// TIA Portal V17 export
// export: Created 2025-03-10T13:12:17.8643549Z, ExportSetting WithDefaults, DisplayName Totally Integrated Automation Portal, DisplayVersion V17 Update 8, DisplayName TIA Portal Openness, DisplayVersion V17 Update 8, DisplayName TIA Portal Version Control Interface, DisplayVersion V17, DisplayName SINAMICS Startdrive Advanced, DisplayVersion V17 SP2, DisplayName SINAMICS Startdrive G110M, G120, G120C, G120D, G120P, G115D, DisplayVersion V17 SP2, DisplayName SINAMICS Startdrive G130, G150, S120, S150, SINAMICS MV, S210, DisplayVersion V17 SP2, DisplayName STEP 7 Professional, DisplayVersion V17 Update 8, DisplayName SINUMERIK ONE STEP 7 Toolbox, DisplayVersion V17 Update 12, DisplayName SINUMERIK 840D sl STEP 7 Toolbox, DisplayVersion V17 Update 12, DisplayName STEP 7 Safety, DisplayVersion V17 Update 6, DisplayName WinCC Advanced, DisplayVersion V17 Update 8
TYPE "FANUC_INPUTS"
// stored: IsFailsafeCompliant false
   STRUCT
      SYSTEM_SIGNAL : Struct
         SYS_IMSTP : Bool;   // MACHINE HEARTBEAT (MACHINE TO GANTRY) / IMMEDIATE STOP
         SYS_HOLD : Bool;   // HOLD ROBOT
         SYS_SFSPD : Bool;   // MACHINE EMERGENCY STOP OK (MACHINE TO GANTRY) / SAFE SPEED
         SYS_CYCLE_STOP : Bool;   // MACHINE SAFETY GATES OK (LOCKED)(MACHINE TO GANTRY) / CYCLE STOP
         SYS_FAULT_RESET : Bool;   // MACHINE IN MANUAL MODE (MACHINE TO GANTRY) / FAULT RESET
         SYS_HOME : Bool;   // MACHINE IN AUTO MODE(MACHINE TO GANTRY) / HOME
         SYS_START : Bool;   // MACHINE AUTO CYCLE RUNNING (MACHINE TO GANTRY) / START PROGRAM / CONTINUE PROGRAM
         SYS_MOTION_ENBL : Bool;   // MACHINE IS IN WARMUP CYCLE (MACHINE TO GANTRY) / MOTION ENABLE
         SPARE_65_0 : Byte;   // MACHINE IN RUN OUT MODE (MACHINE TO GANTRY)
         SPARE_66_0 : Byte;   // MACHINE PART DEMAND SOON (MACHINE TO GANTRY)
         SPARE_67_0 : Byte;
      END_STRUCT;
      GENERAL_SIGNAL : Struct
         STYLE_INIT : Bool;   // GANTRY HEARTBEAT (GANTRY TO MACHINE) / INITIATE STYLE PROGRAM
         READ_DEC_CODE : Bool;   // READ DECISION CODE
         OK_CONTINUE : Bool;   // GANTRY EMERGENCY STOP OK (GANTRY TO MACHINE) / OK TO CONTINUE
         ENTER_REQUEST : Bool;   // ENTER CELL REQUEST
         DRY_CYCLE : Bool;   // GANTRY IN MANUAL MODE (GANTRY TO MACHINE) / DRY CYCLE
         RECOVER_REQ : Bool;   // GANTRY IN AUTO MODE (GANTRY TO MACHINE) / RECOVERY REQUEST
         SPARE_68_6 : Bool;   // GANTRY IN AUTO CYCLE RUNNING (GANTRY TO MACHINE)
         SPARE_68_7 : Bool;   // GANTRY OVERHEAD DOOR CLOSED & LOCKED (GANTRY TO MACHINE)
         IMMEDIATE_STOP_AUX : Bool;
         STOP_END_OF_CYCLE : Bool;
         RUNOUT_REQUEST : Bool;
         SPARE_69_3 : Bool;
         SPARE_69_4 : Bool;
         SPARE_69_5 : Bool;
         SPARE_69_6 : Bool;
         SPARE_69_7 : Bool;
         SPARE_70_0 : Byte;   // GANTRY CLEAR OF MACHINE (GANTRY TO MACHINE)
         SPARE_71_0 : Byte;   // GANTRY CLEAR OF FIXTURE (GANTRY TO MACHINE)
         SPARE_72_0 : Byte;
         SPARE_73_0 : Byte;
      END_STRUCT;
      PROGRAM : Struct
         STYLE_PROGRAM : Byte;   // GANTRY HEARTBEAT (GANTRY TO MACHINE) / GROUP INPUT INDICATING STYLE NUMBER PROGRAM
         DEC_CODE : Byte;   // SPECIFIC OPERATING WITHIN A STYLE
         PART_TYPE : Byte;   // GANTRY EMERGENCY STOP OK (GANTRY TO MACHINE) / PART TYPE SELECTED
         SPARE_77_0 : Byte;   // GANTRY EMERGENCY STOP OK (GANTRY TO MACHINE)
      END_STRUCT;
      GRIPPERS : Struct
         T1_GRIPPER_A_OPEN_REQ : Bool;   // ROBOT TOOL 1 GRIPPER A OPEN REQUEST
         T1_GRIPPER_A_CLOSE_REQ : Bool;   // ROBOT TOOL 1 GRIPPER A CLOSE REQUEST
         SPARE_78_2 : Bool;
         SPARE_78_3 : Bool;
         T1_GRIPPER_A_OPEN : Bool;   // ROBOT TOOL 1 GRIPPER A OPEN
         T1_GRIPPER_A_CLOSED : Bool;   // ROBOT TOOL 1 GRIPPER A CLOSED
         SPARE_78_6 : Bool;
         SPARE_78_7 : Bool;
         T1_GRIPPER_B_OPEN_REQ : Bool;   // ROBOT TOOL 1 GRIPPER B OPEN REQUEST
         T1_GRIPPER_B_CLOSE_REQ : Bool;   // ROBOT TOOL 1 GRIPPER B CLOSE REQUEST
         SPARE_79_2 : Bool;
         SPARE_79_3 : Bool;
         T1_GRIPPER_B_OPEN : Bool;   // ROBOT TOOL 1 GRIPPER B OPEN
         T1_GRIPPER_B_CLOSED : Bool;   // ROBOT TOOL 1 GRIPPER B CLOSED
         SPARE_79_6 : Bool;
         SPARE_79_7 : Bool;
         T1_GRIPPER_C_OPEN_REQ : Bool;   // ROBOT TOOL 1 GRIPPER C OPEN REQUEST
         T1_GRIPPER_C_CLOSE_REQ : Bool;   // ROBOT TOOL 1 GRIPPER C CLOSE REQUEST
         SPARE_80_2 : Bool;
         SPARE_80_3 : Bool;
         T1_GRIPPER_C_OPEN : Bool;   // ROBOT TOOL 1 GRIPPER C OPEN
         T1_GRIPPER_C_CLOSED : Bool;   // ROBOT TOOL 1 GRIPPER C CLOSED
         SPARE_80_6 : Bool;
         SPARE_80_7 : Bool;
         T1_GRIPPER_D_OPEN_REQ : Bool;   // ROBOT TOOL 1 GRIPPER D OPEN REQUEST
         T1_GRIPPER_D_CLOSE_REQ : Bool;   // ROBOT TOOL 1 GRIPPER D CLOSE REQUEST
         SPARE_81_2 : Bool;
         SPARE_81_3 : Bool;
         T1_GRIPPER_D_OPEN : Bool;   // ROBOT TOOL 1 GRIPPER D OPEN
         T1_GRIPPER_D_CLOSED : Bool;   // ROBOT TOOL 1 GRIPPER D CLOSED
         SPARE_81_6 : Bool;
         SPARE_81_7 : Bool;
         T1_GRIPPER_E_OPEN_REQ : Bool;   // ROBOT TOOL 1 GRIPPER E OPEN REQUEST
         T1_GRIPPER_E_CLOSE_REQ : Bool;   // ROBOT TOOL 1 GRIPPER E CLOSE REQUEST
         SPARE_82_2 : Bool;
         SPARE_82_3 : Bool;
         T1_GRIPPER_E_OPEN : Bool;   // ROBOT TOOL 1 GRIPPER E OPEN
         T1_GRIPPER_E_CLOSED : Bool;   // ROBOT TOOL 1 GRIPPER E CLOSED
         SPARE_82_6 : Bool;
         SPARE_82_7 : Bool;
         T2_GRIPPER_A_OPEN_REQ : Bool;   // ROBOT TOOL 2 GRIPPER A OPEN REQUEST
         T2_GRIPPER_A_CLOSE_REQ : Bool;   // ROBOT TOOL 2 GRIPPER A CLOSE REQUEST
         SPARE_83_2 : Bool;
         SPARE_83_3 : Bool;
         T2_GRIPPER_A_OPEN : Bool;   // ROBOT TOOL 2 GRIPPER A OPEN
         T2_GRIPPER_A_CLOSED : Bool;   // ROBOT TOOL 2 GRIPPER A CLOSED
         SPARE_83_6 : Bool;
         SPARE_83_7 : Bool;
         T2_GRIPPER_B_OPEN_REQ : Bool;   // ROBOT TOOL 2 GRIPPER B OPEN REQUEST
         T2_GRIPPER_B_CLOSE_REQ : Bool;   // ROBOT TOOL 2 GRIPPER B CLOSE REQUEST
         SPARE_84_2 : Bool;
         SPARE_84_3 : Bool;
         T2_GRIPPER_B_OPEN : Bool;   // ROBOT TOOL 2 GRIPPER B OPEN
         T2_GRIPPER_B_CLOSED : Bool;   // ROBOT TOOL 2 GRIPPER B CLOSED
         SPARE_84_6 : Bool;
         SPARE_84_7 : Bool;
         T2_GRIPPER_C_OPEN_REQ : Bool;   // ROBOT TOOL 2 GRIPPER C OPEN REQUEST
         T2_GRIPPER_C_CLOSE_REQ : Bool;   // ROBOT TOOL 2 GRIPPER C CLOSE REQUEST
         SPARE_85_2 : Bool;
         SPARE_85_3 : Bool;
         T2_GRIPPER_C_OPEN : Bool;   // ROBOT TOOL 2 GRIPPER C OPEN
         T2_GRIPPER_C_CLOSED : Bool;   // ROBOT TOOL 2 GRIPPER C CLOSED
         SPARE_85_6 : Bool;
         SPARE_85_7 : Bool;
         T2_GRIPPER_D_OPEN_REQ : Bool;   // ROBOT TOOL 2 GRIPPER D OPEN REQUEST
         T2_GRIPPER_D_CLOSE_REQ : Bool;   // ROBOT TOOL 2 GRIPPER D CLOSE REQUEST
         SPARE_86_2 : Bool;
         SPARE_86_3 : Bool;
         T2_GRIPPER_D_OPEN : Bool;   // ROBOT TOOL 2 GRIPPER D OPEN
         T2_GRIPPER_D_CLOSED : Bool;   // ROBOT TOOL 2 GRIPPER D CLOSED
         SPARE_86_6 : Bool;
         SPARE_86_7 : Bool;
         T2_GRIPPER_E_OPEN_REQ : Bool;   // ROBOT TOOL 2 GRIPPER E OPEN REQUEST
         T2_GRIPPER_E_CLOSE_REQ : Bool;   // ROBOT TOOL 2 GRIPPER E CLOSE REQUEST
         SPARE_87_2 : Bool;
         SPARE_87_3 : Bool;
         T2_GRIPPER_E_OPEN : Bool;   // ROBOT TOOL 2 GRIPPER E OPEN
         T2_GRIPPER_E_CLOSED : Bool;   // ROBOT TOOL 2 GRIPPER E CLOSED
         SPARE_87_6 : Bool;
         SPARE_87_7 : Bool;
         T1_ALL_GRIPS_OPEN_REQ : Bool;   // ROBOT TOOL 1 OPEN ALL GRIPPERS REQUEST
         T1_ALL_GRIPS_CLOSE_REQ : Bool;   // ROBOT TOOL 1 CLOSE ALL GRIPPERS REQUEST
         T1_ALL_GRIPPERS_OPEN : Bool;   // ROBOT TOOL 1 ALL GRIPPERS OPEN
         T1_ALL_GRIPPERS_CLOSED : Bool;   // ROBOT TOOL 1 ALL GRIPPERS CLOSED
         SPARE_88_4 : Bool;
         SPARE_88_5 : Bool;
         SPARE_88_6 : Bool;
         SPARE_88_7 : Bool;
         T2_ALL_GRIPS_OPEN_REQ : Bool;   // ROBOT TOOL 2 CLOSE ALL GRIPPERS REQUEST
         T2_ALL_GRIPS_CLOSE_REQ : Bool;   // ROBOT TOOL 2 CLOSE ALL GRIPPERS REQUEST
         T2_ALL_GRIPPERS_OPEN : Bool;   // ROBOT TOOL 2 ALL GRIPPERS OPEN
         T2_ALL_GRIPPERS_CLOSED : Bool;   // ROBOT TOOL 2 ALL GRIPPERS CLOSED
         SPARE_89_4 : Bool;
         SPARE_89_5 : Bool;
         SPARE_89_6 : Bool;
         SPARE_89_7 : Bool;
         SPARE_90_0 : Byte;
         FAULT_NUMBER : Byte;   // FAULT RESPONSE
      END_STRUCT;
      CLEARS : Struct
         CLEAR_U_1 : Bool;   // GANTRY HEARTBEAT (GANTRY TO MACHINE) / CLEAR TO GET IN UNIT 1
         CLEAR_U_2 : Bool;   // CLEAR TO GET IN UNIT 2
         CLEAR_U_3 : Bool;   // GANTRY EMERGENCY STOP OK (GANTRY TO MACHINE) / CLEAR TO GET IN UNIT 3
         CLEAR_U_4 : Bool;   // CLEAR TO GET IN UNIT 4
         CLEAR_U_5 : Bool;   // GANTRY IN MANUAL MODE (GANTRY TO MACHINE) / CLEAR TO GET IN UNIT 5
         CLEAR_U_6 : Bool;   // GANTRY IN AUTO MODE (GANTRY TO MACHINE) / CLEAR TO GET IN UNIT 6
         CLEAR_U_7 : Bool;   // GANTRY IN AUTO CYCLE RUNNING (GANTRY TO MACHINE) / CLEAR TO GET IN UNIT 7
         CLEAR_U_8 : Bool;   // GANTRY OVERHEAD DOOR CLOSED & LOCKED (GANTRY TO MACHINE) / CLEAR TO GET IN UNIT 8
         CLEAR_U_9 : Bool;   // GANTRY IN RUN OUT COMPLETE(GANTRY TO MACHINE) / CLEAR TO GET IN UNIT 9
         CLEAR_U_10 : Bool;   // GANTRY CLEAR OF MACHINE (GANTRY TO MACHINE) / CLEAR TO GET IN UNIT 10
         SPARE_93_2 : Bool;   // GANTRY CLEAR OF FIXTURE (GANTRY TO MACHINE)
         SPARE_93_3 : Bool;
         SPARE_93_4 : Bool;
         SPARE_93_5 : Bool;   // GANTRY PART TYPE CHANGE REQUESTED (GANTRY TO MACHINE)
         SPARE_93_6 : Bool;   // GANTRY REQUEST MACHINE TO RUN WITH LOADED PARTS (GANTRY TO MACHINE)
         SPARE_93_7 : Bool;   // GANTRY RUN OUT REQUESTED (GANTRY TO MACHINE)
         SPARE_94_0 : Byte;
         SPARE_95_0 : Byte;
      END_STRUCT;
      TASKS : Struct
         COMPLETE_TSK_1 : Bool;   // GANTRY HEARTBEAT (GANTRY TO MACHINE) / PICK REQUEST - ST1
         COMPLETE_TSK_2 : Bool;   // PLACE REQUEST - ST1
         COMPLETE_TSK_3 : Bool;   // GANTRY EMERGENCY STOP OK (GANTRY TO MACHINE) / PICK&PLACE REQUEST - ST1
         COMPLETE_TSK_4 : Bool;   // ROBOT COMPLETE TASK 4
         COMPLETE_TSK_5 : Bool;   // GANTRY IN MANUAL MODE (GANTRY TO MACHINE) / ROBOT COMPLETE TASK 5
         COMPLETE_TSK_6 : Bool;   // GANTRY IN AUTO MODE (GANTRY TO MACHINE) / ROBOT COMPLETE TASK 6
         COMPLETE_TSK_7 : Bool;   // GANTRY IN AUTO CYCLE RUNNING (GANTRY TO MACHINE) / ROBOT COMPLETE TASK 7
         COMPLETE_TSK_8 : Bool;   // GANTRY OVERHEAD DOOR CLOSED & LOCKED (GANTRY TO MACHINE) / ROBOT COMPLETE TASK 8
         SPARE_97_0 : Byte;   // GANTRY IN RUN OUT COMPLETE(GANTRY TO MACHINE)
         SPARE_98_0 : Byte;   // GANTRY CLEAR OF MACHINE (GANTRY TO MACHINE)
         SPARE_99_0 : Byte;   // GANTRY CLEAR OF FIXTURE (GANTRY TO MACHINE)
         SPARE_100_0 : Byte;
         SPARE_101_0 : Byte;
         SPARE_102_0 : Byte;
         SPARE_103_0 : Byte;
      END_STRUCT;
      PARTS_ENABLED : Struct
         PART_A_ENABLED : Bool;   // GANTRY HEARTBEAT (GANTRY TO MACHINE) / PART A ENABLED TO WORK
         PART_B_ENABLED : Bool;   // PART B ENABLED TO WORK
         PART_C_ENABLED : Bool;   // GANTRY EMERGENCY STOP OK (GANTRY TO MACHINE) / PART C ENABLED TO WORK
         PART_D_ENABLED : Bool;   // PART D ENABLED TO WORK
         PART_E_ENABLED : Bool;   // GANTRY IN MANUAL MODE (GANTRY TO MACHINE) / PART E ENABLED TO WORK
         SPARE_104_5 : Bool;   // GANTRY IN AUTO MODE (GANTRY TO MACHINE)
         SPARE_104_6 : Bool;   // GANTRY IN AUTO CYCLE RUNNING (GANTRY TO MACHINE)
         SPARE_104_7 : Bool;   // GANTRY OVERHEAD DOOR CLOSED & LOCKED (GANTRY TO MACHINE)
         SPARE_105_0 : Byte;   // GANTRY CLEAR OF FIXTURE (GANTRY TO MACHINE)
      END_STRUCT;
      SPARES : Array[106..127] of Byte;
   END_STRUCT;
END_TYPE
